(* PLC project OOP_Curso, Beckhoff Automation GmbH TwinCAT PLC Control 3.5.13.21 *)
(* stored: creationDateTime 2023-08-10T12:11:53.3599867, modificationDateTime 2023-08-10T12:11:53.3668192 *)

INTERFACE I_Mover
METHOD Mover : REAL
VAR_INPUT
	Velocidad_Deseada : REAL;
END_VAR
END_METHOD
END_INTERFACE

FUNCTION_BLOCK Coche1 EXTENDS Vehiculo
VAR_INPUT
	velocidadMaxima : REAL;
END_VAR
VAR_OUTPUT
END_VAR
VAR
END_VAR

            
          

METHOD Mover : REAL
VAR_INPUT
	Velocidad_Deseada : REAL;
END_VAR
                  Mover := Velocidad_Deseada * velocidadMaxima;
                
END_METHOD
END_FUNCTION_BLOCK

FUNCTION_BLOCK Conductor
VAR_INPUT
	vehiculo : REFERENCE TO Vehiculo(THIS^); // referencia a la clase base Vehiculo
END_VAR
VAR_OUTPUT
END_VAR
VAR
END_VAR

            
          

METHOD Mover : REAL
VAR_INPUT
	Velocidad_Deseada : REAL;
END_VAR
                  Mover := THIS^.vehiculo.Mover(Velocidad_Deseada);

                
END_METHOD
END_FUNCTION_BLOCK

FUNCTION_BLOCK Moto1 EXTENDS Vehiculo
VAR_INPUT
	Aceleracion : REAL;
END_VAR
VAR_OUTPUT
END_VAR
VAR
END_VAR

            
          

METHOD Mover : REAL
VAR_INPUT
	Velocidad_Deseada : REAL;
END_VAR
                  Mover := Velocidad_Deseada * Aceleracion ;
                
END_METHOD
END_FUNCTION_BLOCK

FUNCTION_BLOCK Vehiculo IMPLEMENTS I_Mover

            
          

METHOD Mover : REAL
VAR_INPUT
	Velocidad_Deseada : REAL;
END_VAR
                  Mover := Velocidad_Deseada;
                
END_METHOD
END_FUNCTION_BLOCK

PROGRAM _26_SOLID_LSP
VAR
	Audi_A8 : Coche1;
	Audi_A8_Velocidad_Desada :REAL;
	Audi_A8_Velocidad :REAL;
	
	Suzuki_Ninja: Moto1;
	Suzuki_Ninja_Velocidad_Deseada :REAL;
	Suzuki_Ninja_Velocidad :REAL;
	
	Conductor_Juan : Conductor;
	Conductor_Juan_Velocidad_Deseada :REAL;
	Conductor_Juan_Velocidad : REAL;
	Vehiculo_Seleccionado_Audi_A8 : BOOL;
END_VAR

            Audi_A8_Velocidad := Audi_A8.Mover(Audi_A8_Velocidad_Desada);

Suzuki_Ninja_Velocidad := Suzuki_Ninja.Mover(Suzuki_Ninja_Velocidad_Deseada);

IF Vehiculo_Seleccionado_Audi_A8 = TRUE THEN
	Conductor_Juan(vehiculo:= Audi_A8);
ELSE
	Conductor_Juan(vehiculo:= Suzuki_Ninja);
END_IF

Conductor_Juan_Velocidad := Conductor_Juan.Mover(Conductor_Juan_Velocidad_Deseada);
          
END_PROGRAM
